FUNCTION_BLOCK adsCommunication IMPLEMENTS ITF_ReportDataTool
VAR_INPUT
END_VAR
VAR_OUTPUT
END_VAR
VAR
END_VAR

METHOD Report : BOOL
VAR_INPUT
	somemessage : ARRAY[0..5] OF BYTE;
END_VAR
END_METHOD

END_FUNCTION_BLOCK

(* stored: Version 1.1.0.1, ProductVersion 3.1.4024.12
   POU adsCommunication: Id {2e5f369c-00b9-4463-852a-b63ad1f6bae6}, SpecialFunc None
   Method Report: Id {8b03de4e-b985-45c4-b193-670cfc500963} *)
